TYPE  ST_SoftSettings_Genset:
STRUCT
	b_AutoStartStop						: BOOL;
	b_HydridMode						: BOOL;
	b_EnableSchedule					: BOOL;
	//General settings
	setpointTimeslot1					: ST_Genset_setpoints;
	setpointTimeslot2					: ST_Genset_setpoints;
	b_PSBExtGensetMonitoring			: BOOL; //FUTURE WORK, use PSB to monitor ext fixed power genset.
	b_FreqProtectionEnable				: BOOL;
	Generator 							: ST_Genset_params;
	Loadbank							: ST_Loadbank_params;
END_STRUCT
END_TYPE

(* stored: Version 1.1.0.1, ProductVersion 3.1.4026.18
   DUT ST_SoftSettings_Genset: Id {75cbb5ef-48be-464c-9747-4ba476ebadba} *)
